{attribute 'linkalways'}
{attribute 'no_explicit_call' := 'do not call this POU directly'}
{attribute 'reflection'}
{attribute 'enable_dynamic_creation'}
FUNCTION_BLOCK Instance IMPLEMENTS I_Instance, I_Collectable
{attribute 'hide_all_locals'}
VAR
	{attribute 'instance-path'} 
    {attribute 'noinit'} 
	instancePath : T_MAXSTRING;
	instanceNamespace : STRING := GetNamespace();
	globalNamespace : GlobalNamespace(THIS^);
END_VAR

METHOD PRIVATE GetNamespace : STRING
IF InstancePathIsFilled() THEN
	GetNamespace := ReturnNamespaceFromInstancePath(instancePath);
	RETURN;
END_IF

IF IsNewObjectDuringInitialization() THEN
	GetNamespace := globalNamespace.GetLastInstanceNamespace();
END_IF
END_METHOD

METHOD PRIVATE InstancePathIsFilled : BOOL
InstancePathIsFilled := instancePath <> '';
END_METHOD

METHOD PRIVATE IsNewObjectDuringInitialization : BOOL
VAR CONSTANT 
	PLC_INIT_PHASE : INT := 0;
END_VAR
IsNewObjectDuringInitialization := GETCURTASKINDEXEX() = PLC_INIT_PHASE;
END_METHOD

PROPERTY PUBLIC NameSpace : STRING
GET
Namespace := instanceNamespace;
END_GET
END_PROPERTY

METHOD PUBLIC SharesNamespaceWith : BOOL
VAR_INPUT
	OtherInstance : I_Instance;
END_VAR
SharesNamespaceWith := (Namespace = OtherInstance.NameSpace);
END_METHOD

END_FUNCTION_BLOCK

(* stored: Version 1.1.0.1, ProductVersion 3.1.4024.11
   POU Instance: Id {61104ee8-d822-48ac-bc47-45dfd009ac1e}, SpecialFunc None
   Folder Internal: Id {76b2da4f-a3ed-429e-bbe9-ef5156816628}
   Method GetNamespace: Id {e810ce99-9d71-40ac-ae11-a84e6012dcad}
   Method InstancePathIsFilled: Id {a2b17ef6-cb9e-476e-9f89-78e97494c366}
   Method IsNewObjectDuringInitialization: Id {f91ae77a-c70e-4c49-b9e0-7278c8ae9b64}
   Property NameSpace: Id {7ae71e18-c030-4e06-a315-882f3a357dc0}
   Get Get: Id {c3db41fa-c4f3-4c5f-9e86-90343b017ae9}
   Method SharesNamespaceWith: Id {8bc887fe-eaed-4854-bdd7-2e4b9a46a836} *)
